PROGRAM P_ControlBox
VAR
	fbControlBox : FB_ControlBox; 
	bRealControlBox : BOOL := TRUE;
END_VAR

fbControlBox(
bRealControlBox := bRealControlBox,
eStatus := G_Work.eStatus,
eMode => G_Work.eMode,
);

END_PROGRAM

(* stored: Version 1.1.0.1, ProductVersion 3.1.4024.13
   POU P_ControlBox: Id {f099b577-7c17-4f98-8e29-157282967496}, SpecialFunc None *)
